(* PLC project  *)

PROGRAM ArrayRepeatLimit
  VAR
    Values : ARRAY[1..2] OF INT := [1000001(1)];
  END_VAR

END_PROGRAM
